(* CoDeSys 2.3 export: TANALOGOUTPUT.EXP *)

(* Data type *)
TYPE tAnalogOutput : REAL;
END_TYPE
